// TwinCAT 3 PLC project MyDailyRoutine
// ProgramVersion: 3.1.4024.0
// libraries:
//   Tc2_Standard, * (Beckhoff Automation GmbH)
//   Tc2_System, * (Beckhoff Automation GmbH)
//   Tc3_Module, * (Beckhoff Automation GmbH)
// project tree:
//   / ElevatorTask_1.TcTTO, MorningBreakfast.TcTTO
//   GVLs/ GVL.TcGVL
//   POUs/ ElevatorFunction.TcPOU, ElevatorTask.TcPOU, MormingBreakfastTask.TcPOU
// real-time tasks:
//   TASK MorningBreakfast: cycle T#10ms, priority 1, ADS port 351
//   TASK ElevatorTask: cycle T#5ms, priority 2, ADS port 352

CONFIGURATION MyDailyRoutine
    RESOURCE PLC ON TwinCAT3
        TASK ElevatorTask_1(INTERVAL := T#5ms, PRIORITY := 2);
        TASK MorningBreakfast(INTERVAL := T#10ms, PRIORITY := 1);
        PROGRAM ElevatorTask WITH ElevatorTask_1 : ElevatorTask;
        PROGRAM MormingBreakfastTask WITH MorningBreakfast : MormingBreakfastTask;
    END_RESOURCE
END_CONFIGURATION

// ---- GVLs/GVL.TcGVL
{attribute 'qualified_only'}
VAR_GLOBAL
	bGetUp : BOOL := TRUE;
	bReady : BOOL;
END_VAR

// ---- POUs/ElevatorTask.TcPOU
PROGRAM ElevatorTask
VAR
	//Varibles booleans
	bAllPrepared 		: BOOL;
	bPressButton 		: BOOL;
	bElevatorArrives 	: BOOL;
	bEnterElevator 		: BOOL;
	bPressFirstFloor	: BOOL;
	bCheckClass 		: BOOL;
	bGoToUniversity 	: BOOL;
	bGoToGym			: BOOL;
	bDone				: BOOL;
	//Variables timers	
	fbGoToElevator 		: TON;
	fbWaitElevator 		: TON;
	fbGoToFirstFloor 	: TON;
	fbWalkToUniversity	: TON;
	fbWalkToClassroom	: TON;
END_VAR

//First step: When i finish my breakfast i prepare my thing and go to take the elevator
	IF GVL.bReady THEN
		bAllPrepared := TRUE;
		fbGoToElevator(IN:=bAllPrepared,PT:=T#3S);
	END_IF

	IF fbGoToElevator.Q THEN
		bPressButton := TRUE;
		fbWaitElevator(IN:=bPressButton,PT:=T#3S);
	END_IF
	
	IF fbWaitElevator.Q THEN
		bElevatorArrives := TRUE;
		bEnterElevator :=bElevatorArrives;
		bPressFirstFloor := bEnterElevator;
		fbGoToFirstFloor(IN:=bPressFirstFloor,PT:=T#4S);
	END_IF
//Second step: When im in the first floor i decide where i want to go

	bCheckClass := ElevatorFunction(bCheckClass := fbGoToFirstFloor.Q);		//Function
	
	IF bCheckClass THEN
		bGoToUniversity := TRUE;
		bGoToGym := FALSE;
	ELSE
		bGoToUniversity := FALSE;
		bGoToGym := TRUE;
	END_IF

//Third step: Go to university and classroom

	fbWalkToUniversity(IN:=bGoToUniversity,PT:=T#5S);
	fbWalkToClassroom(IN:=fbWalkToUniversity.Q,PT:=T#5S);
	
	bDone := fbWalkToClassroom.Q;											//Me in classroom

END_PROGRAM

// ---- POUs/ElevatorFunction.TcPOU
FUNCTION ElevatorFunction : BOOL

VAR_INPUT
	bCheckClass 	: BOOL;
END_VAR

VAR
	bMyDecision : BOOL;
END_VAR

IF bCheckClass THEN
	ElevatorFunction := TRUE;
ELSE
	ElevatorFunction := FALSE;
END_IF

END_FUNCTION

// ---- POUs/MormingBreakfastTask.TcPOU
PROGRAM MormingBreakfastTask
VAR
	//Variables booleans
	bHungry 			: BOOL;
	bStartPreparation 	: BOOL;
	bStartEat 			: BOOL;
	bReady 				: BOOL;
	//Variables timers
	fbGoToKitchen 		: TON;
	fbDecideIfIEat 		: TON;
	fbPrepareTea 		: TON;
	fbPrepareEggs 		: TON;
	fbPrepareBread 		: TON;
	fbImEating 			: TON;
END_VAR

//First step: Get up and decide if want to eat breakfast

fbDecideIfIEat(IN:=GVL.bGetUp,PT:=T#3S);

IF fbDecideIfIEat.Q THEN
	bHungry := TRUE;
END_IF
fbGoToKitchen(IN:=bHungry,PT:=T#3S);

//Second Step: Now in the kitchen im going to prepare my breakfast

IF fbGoToKitchen.Q THEN
	bStartPreparation := TRUE;
END_IF

fbPrepareTea(IN:=bStartPreparation,PT:=T#7S);     //Im going to use this .Q because it is the last to finish when i cook
fbPrepareBread(IN:=bStartPreparation,PT:=T#3S);
fbPrepareEggs(IN:=bStartPreparation,PT:=T#5S);

//Third step: Finally i end the preparation and start to eat

IF fbPrepareTea.Q AND NOT bStartEat THEN
    bStartEat := TRUE;
END_IF

fbImEating(IN := bStartEat, PT := T#10S);

GVL.bReady := fbImEating.Q;

END_PROGRAM
